(* Logix 5000 project; controller ZaxisVmpEdsSample vendor 1 type 14 code 196 rev 33.11; software revision 33.00 *)

TASK MainTask (continuous, watchdog 500 ms) : MainProgram, Vmp_Interface

MODULES
   Local : vendor 1 type 14 code 196 (5069 0, rev 33.11)
      Inputs : 5069-IB16 (5069 1, rev 2.1, StandardDataDriven RPI 5 ms)
      Outputs : vendor 1 type 7 code 396 (5069 2, rev 2.1, StandardDataDriven RPI 5 ms)
      Vmp_00 : vendor 1449 type 43 code 17 (Ethernet 192.168.2.130, rev 1.4, StandardDataDriven RPI 500 ms)
END_MODULES

TYPE STRING_12 :
STRUCT
   LEN : DINT;
   DATA : SINT[12];
END_STRUCT
END_TYPE

TYPE STRING_16_UDT :
STRUCT
   LEN : DINT;
   DATA : SINT[16];
END_STRUCT
END_TYPE

TYPE STRING_20 :
STRUCT
   LEN : DINT;
   DATA : SINT[20];
END_STRUCT
END_TYPE

TYPE STRING_24 :
STRUCT
   LEN : DINT;
   DATA : SINT[24];
END_STRUCT
END_TYPE

TYPE Vmp_Config :
STRUCT
   CosType : INT;   // Change-of-State Type
   ClassId : INT;   // ClassId
   Instance : INT;   // Instance
   Attribute : INT;   // Attribute
   CfgVersion : INT;   // CfgVersion
   CfgLength : INT;   // CfgLength
   NumberOfHeads : SINT;   // NumberOfHeads
   PumpType : SINT;   // PumpType
   PumpNumber : SINT;   // PumpNumber
   HeadSize : SINT;   // HeadSize
   AdjustStepmode : INT;   // AdjustStepmode
   ZinchRpm : INT;   // ZinchRpm
   Baud : INT;   // Baud
   ExtraSteps : INT;   // ExtraSteps
   SpareInt1 : INT;   // SpareInt1
   SpareInt2 : INT;   // SpareInt2
   ReadyInterlock : BOOL;   // ReadyInterlock
   EthernetRunReady : BOOL;   // EthernetRunReady
   DchpEnabled : BOOL;   // DchpEnabled
   BoreInCm : BOOL;   // BoreInCm
   IoStartFallingEdge : BOOL;   // IoStartFallingEdge
   FullDuplexRs485 : BOOL;   // FullDuplexRs485
   Spare1_6 : BOOL;   // Spare1_6
   IsFinePichAdj : BOOL;   // IsFinePichAdj
   Spare1_8 : BOOL;   // Spare1_8
   Spare1_9 : BOOL;   // Spare1_9
   Spare1_10 : BOOL;   // Spare1_10
   Spare1_11 : BOOL;   // Spare1_11
   Spare1_12 : BOOL;   // Spare1_12
   Spare1_13 : BOOL;   // Spare1_13
   Spare1_14 : BOOL;   // Spare1_14
   Spare1_15 : BOOL;   // Spare1_15
   Spare1_16 : BOOL;   // Spare1_16
   Spare1_17 : BOOL;   // Spare1_17
   Spare1_18 : BOOL;   // Spare1_18
   Spare1_19 : BOOL;   // Spare1_19
   Spare1_20 : BOOL;   // Spare1_20
   Spare1_21 : BOOL;   // Spare1_21
   Spare1_22 : BOOL;   // Spare1_22
   Spare1_23 : BOOL;   // Spare1_23
   IsServo : BOOL;   // IsServo
   OkToResetDevice : BOOL;   // OkToResetDevice
   Spare1_26 : BOOL;   // Spare1_26
   Spare1_27 : BOOL;   // Spare1_27
   Spare1_28 : BOOL;   // Spare1_28
   Spare1_29 : BOOL;   // Spare1_29
   Spare1_30 : BOOL;   // Spare1_30
   Spare1_31 : BOOL;   // Spare1_31
   FirmwareRev : DINT;   // FirmwareRev
   Bore : DINT;   // Bore
   OffsetValue : DINT;   // OffsetValue
   FlashWriteCnt : DINT;   // FlashWriteCnt
   FaultDispenseSensorCnt : DINT;   // FaultDispenseSensorCnt
   FaultDispenseMotorCnt : DINT;   // FaultDispenseMotorCnt
   FaultAdjustSensorCnt : DINT;   // FaultAdjustSensorCnt
   FaultAdjustMotorCnt : DINT;   // FaultAdjustMotorCnt
   SpareDInt1 : DINT;   // SpareDInt1
   SpareDint2 : DINT;   // SpareDint2
   SerialNumber : STRING_16_UDT;   // SerialNumber
   IpAddress : STRING_16_UDT;   // IpAddress
   IpNetmask : STRING_16_UDT;   // IpNetmask
   IpGateway : STRING_16_UDT;   // IpGateway
   MacAddress : STRING_20;   // MacAddress
   ModelNumber : STRING_24;   // ModelNumber
   OptionsAndFittings : STRING_24;   // OptionsAndFittings
   SccsRevDate : STRING_24;   // SccsRevDate
   SccsRev : STRING_12;   // SccsRev
   SccsRevRange : STRING_24;   // SccsRevRange
END_STRUCT
END_TYPE

TYPE VMP_Program :
STRUCT
   CosType : INT;   // CosType
   ClassId : INT;   // ClassId
   Instance : INT;   // Instance
   Attribute : INT;   // Attribute
   CfgVersion : INT;   // CfgVersion
   CfgLength : INT;   // CfgLength
   Direction : BOOL;   // Direction
   ContinuousRun : BOOL;   // ContinuousRun
   Spare1_2 : BOOL;   // Spare1_2
   Spare1_3 : BOOL;   // Spare1_3
   Spare1_4 : BOOL;   // Spare1_4
   Spare1_5 : BOOL;   // Spare1_5
   Spare1_6 : BOOL;   // Spare1_6
   Spare1_7 : BOOL;   // Spare1_7
   Spare1_8 : BOOL;   // Spare1_8
   Spare1_9 : BOOL;   // Spare1_9
   Spare1_10 : BOOL;   // Spare1_10
   Spare1_11 : BOOL;   // Spare1_11
   Spare1_12 : BOOL;   // Spare1_12
   Spare1_13 : BOOL;   // Spare1_13
   Spare1_14 : BOOL;   // Spare1_14
   Spare1_15 : BOOL;   // Spare1_15
   Spare1_16 : BOOL;   // Spare1_16
   Spare1_17 : BOOL;   // Spare1_17
   Spare1_18 : BOOL;   // Spare1_18
   Spare1_19 : BOOL;   // Spare1_19
   Spare1_20 : BOOL;   // Spare1_20
   Spare1_21 : BOOL;   // Spare1_21
   Spare1_22 : BOOL;   // Spare1_22
   Spare1_23 : BOOL;   // Spare1_23
   Spare1_24 : BOOL;   // Spare1_24
   Spare1_25 : BOOL;   // Spare1_25
   Spare1_26 : BOOL;   // Spare1_26
   Spare1_27 : BOOL;   // Spare1_27
   Spare1_28 : BOOL;   // Spare1_28
   Spare1_29 : BOOL;   // Spare1_29
   Spare1_30 : BOOL;   // Spare1_30
   Spare1_31 : BOOL;   // Spare1_31
   ProgramNumber : INT;   // ProgramNumber
   PullBack : INT;   // PullBack
   PullBackRpm : INT;   // PullBackRpm
   PullBackEndCycleRpm : INT;   // PullBackEndCycleRpm
   PullBackEndCycle : INT;   // PullBackEndCycle
   PullBackEndCycleDelay : INT;   // PullBackEndCycleDelay
   InitialRpm : INT;   // InitialRpm
   Rpm : INT;   // Rpm
   FinalRpm : INT;   // FinalRpm
   FineAdjust : INT;   // FineAdjust
   Acceleration : INT;   // Acceleration
   Deceleration : INT;   // Deceleration
   LoopCycles : INT;   // LoopCycles
   LinkedProgram : INT;   // LinkedProgram
   LinkedTimeDelay : INT;   // LinkedTimeDelay
   MotorCurrent : INT;   // MotorCurrent
   Revolutions : INT;   // Revolutions
   PrePumpClamp : INT;   // PrePumpClamp
   PostPumpClamp : INT;   // PostPumpClamp
   AdjInitialRpm : INT;   // AdjInitialRpm
   AdjustRpm : INT;   // AdjustRpm
   AdjustAcceleration : INT;   // AdjustAcceleration
   AdjustDeceleration : INT;   // AdjustDeceleration
   AdjustMotorPwr : INT;   // AdjustMotorPwr
   SpareInt1 : INT;   // SpareInt1
   SpareInt2 : INT;   // SpareInt2
   AdjustMotorSteps : DINT;   // AdjustMotorSteps
   ApproxDispenseTime : DINT;   // ApproxDispenseTime
   Volume : REAL;   // Volume
   SpareDint1 : REAL;   // SpareDint1
   ProgramName : STRING_16_UDT;   // ProgramName
END_STRUCT
END_TYPE

TYPE Vmp_Pump :
STRUCT
   Enabled : BOOL;
   State : INT;   // Current State
   ShotCount : DINT;   // Number of shots
   DisconnectCount : DINT;   // Disconnect Counter
   FaultCount : DINT;   // Fault Counter
   IN : _05A9:VMP_1_4_21408F44:I:0;
   OUT : _05A9:VMP_1_4_0C80E81B:O:0;
   Configuration : Vmp_Config;
   Programs : VMP_Program[50];
   PumpTmr : TIMER;   // Used to time prime and/or zinch mode
END_STRUCT
END_TYPE

TYPE VMP_Setup :
STRUCT
   ReadyInterlock : BOOL;   // RdyInputEnabled
   EthernetRunReady : BOOL;   // EthSendBusy
   HoldOnFault : BOOL;   // HoldOnFault
   Spare1_3 : BOOL;   // Spare Bit
   Spare1_4 : BOOL;   // Spare Bit
   Spare1_5 : BOOL;   // Spare Bit
   Spare1_6 : BOOL;   // Spare Bit
   Spare1_7 : BOOL;   // Spare Bit
   Spare1_8 : BOOL;   // Spare Bit
   Spare1_9 : BOOL;   // Spare Bit
   Spare1_10 : BOOL;   // Spare Bit
   Spare1_11 : BOOL;   // Spare Bit
   Spare1_12 : BOOL;   // Spare Bit
   Spare1_13 : BOOL;   // Spare Bit
   Spare1_14 : BOOL;   // Spare Bit
   Spare1_15 : BOOL;   // Spare Bit
   Spare1_16 : BOOL;   // Spare Bit
   Spare1_17 : BOOL;   // Spare Bit
   Spare1_18 : BOOL;   // Spare Bit
   Spare1_19 : BOOL;   // Spare Bit
   Spare1_20 : BOOL;   // Spare Bit
   Spare1_21 : BOOL;   // Spare Bit
   Spare1_22 : BOOL;   // Spare Bit
   Spare1_23 : BOOL;   // Spare Bit
   Spare1_24 : BOOL;   // Spare Bit
   Spare1_25 : BOOL;   // Spare Bit
   Spare1_26 : BOOL;   // Spare Bit
   Spare1_27 : BOOL;   // Spare Bit
   Spare1_28 : BOOL;   // Spare Bit
   Spare1_29 : BOOL;   // Spare Bit
   Spare1_30 : BOOL;   // Spare Bit
   Spare1_31 : BOOL;   // Spare Bit
   Baud : DINT;   // Baud
   PumpNumber : DINT;   // PumpNumber
   SpareDInt0 : DINT;   // SpareDInt0
   SpareDInt1 : DINT;   // SpareDInt1
   FirmwareRev : REAL;   // FirmRev
   Bore : REAL;   // Bore
   SpareReal0 : REAL;   // SpareReal0
   SpareReal1 : REAL;   // SpareReal1
   SerialNumber : STRING;   // SerialNumber
END_STRUCT
END_TYPE

TYPE VMP_TcpIP_Cfg :
STRUCT
   Status : DINT;   // Status
   Config_Capability : DINT;   // Capability
   Config_Control : DINT;   // IfCtrl
   Path_Size : INT;   // Epath
   Path : SINT[4];   // Padd
   IP_Address : DINT;   // IPAddr
   Network_Address : DINT;   // NetAddr
   Gateway_Address : DINT;   // GateWay
   Name_Server : DINT;   // DNS1
   Name_Server_2 : DINT;   // DNS2
   Domain_Name : STRING;   // Domain
   Host_Name : STRING;   // Host
   Safety_Network_Number : SINT[6];   // Ignore
   TTL : SINT;   // TTL
   Alloc_Control : SINT;   // MultCast
   Reserved : SINT;   // Reserved
   Num_Mcast : INT;   // MultCastAlloc
   Mcast_Start_Addr : DINT;   // MultCastStart
   Selected_Acd : BOOL;   // ACD
   Acd_Activity : SINT;   // ACDState
   Remote_MAC : SINT[6];   // MACRmt
   Arp_Pdu : SINT[28];   // ARP_PDU
   EthernetIP_Quick_Connect : BOOL;   // QuickCon
   Encp_Inactivity_Timeout : INT;   // InactTimeout
END_STRUCT
END_TYPE

ADD_ON_INSTRUCTION Vmp_Run_Pump   (* revision 1.0 *)
VAR_IN_OUT
   Pump : Vmp_Pump; {required}
END_VAR
VAR_INPUT
   State : INT; {required}
   ShotCount : DINT; {required}
   PrimeRevs : DINT; {required}
   ZinchTime : DINT; {required}
END_VAR
VAR
   DirectionONS : BOOL; {access None}
END_VAR

ROUTINE Logic   (* ladder *)
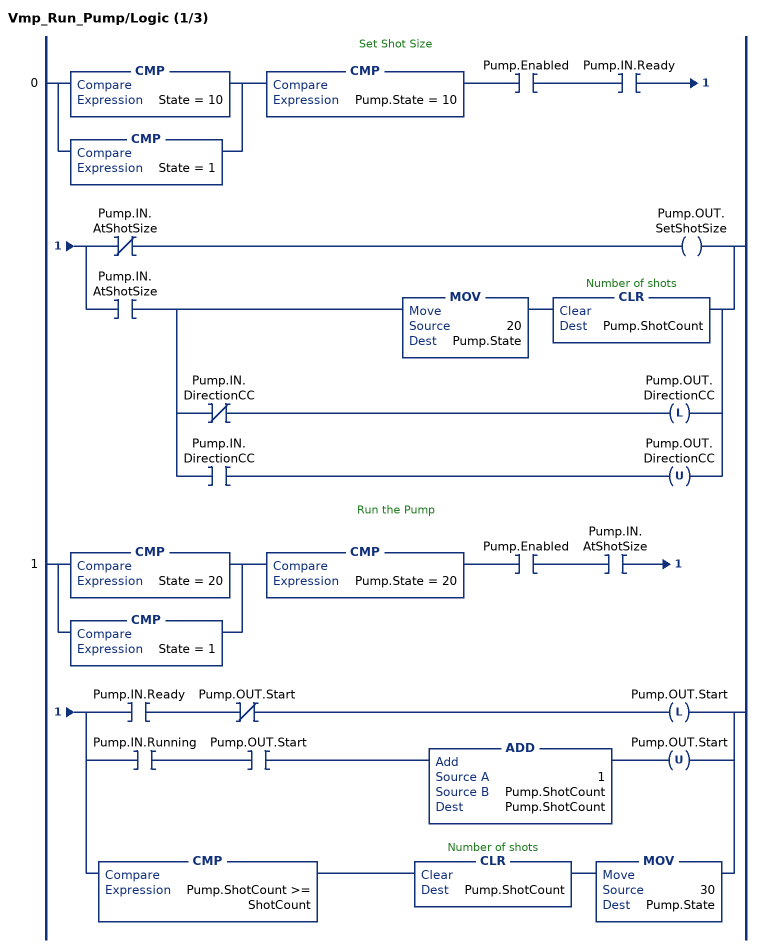
   // Set Shot Size
   0: [CMP(State = 10) ,CMP(State = 1) ]CMP(Pump.State = 10)XIC(Pump.Enabled)XIC(Pump.IN.Ready)[XIO(Pump.IN.AtShotSize) OTE(Pump.OUT.SetShotSize) ,XIC(Pump.IN.AtShotSize) [MOV(20,Pump.State) CLR(Pump.ShotCount) ,XIO(Pump.IN.DirectionCC) OTL(Pump.OUT.DirectionCC) ,XIC(Pump.IN.DirectionCC) OTU(Pump.OUT.DirectionCC) ] ];
   // Run the Pump
   1: [CMP(State = 20) ,CMP(State = 1) ]CMP(Pump.State = 20)XIC(Pump.Enabled)XIC(Pump.IN.AtShotSize)[XIC(Pump.IN.Ready) XIO(Pump.OUT.Start) OTL(Pump.OUT.Start) ,XIC(Pump.IN.Running) XIC(Pump.OUT.Start) ADD(1,Pump.ShotCount,Pump.ShotCount) OTU(Pump.OUT.Start) ,CMP(Pump.ShotCount >= ShotCount) CLR(Pump.ShotCount) MOV(30,Pump.State) ];
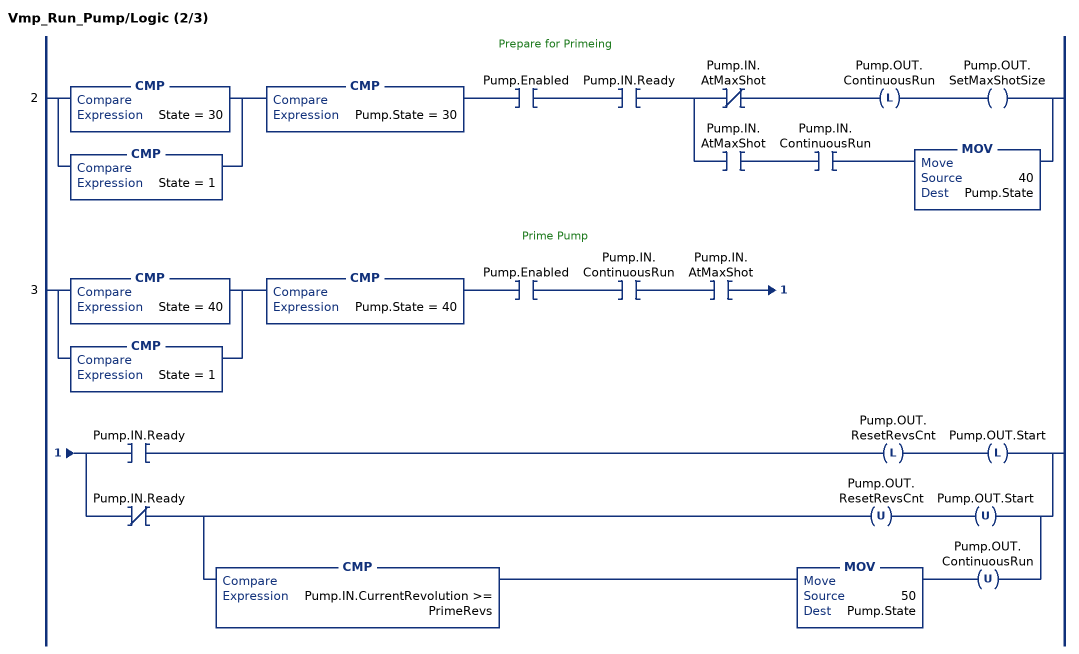
   // Prepare for Primeing
   2: [CMP(State = 30) ,CMP(State = 1) ]CMP(Pump.State = 30)XIC(Pump.Enabled)XIC(Pump.IN.Ready)[XIO(Pump.IN.AtMaxShot) OTL(Pump.OUT.ContinuousRun) OTE(Pump.OUT.SetMaxShotSize) ,XIC(Pump.IN.AtMaxShot) XIC(Pump.IN.ContinuousRun) MOV(40,Pump.State) ];
   // Prime Pump
   3: [CMP(State = 40) ,CMP(State = 1) ]CMP(Pump.State = 40)XIC(Pump.Enabled)XIC(Pump.IN.ContinuousRun)XIC(Pump.IN.AtMaxShot)[XIC(Pump.IN.Ready) OTL(Pump.OUT.ResetRevsCnt) OTL(Pump.OUT.Start) ,XIO(Pump.IN.Ready) [OTU(Pump.OUT.ResetRevsCnt) OTU(Pump.OUT.Start) ,CMP(Pump.IN.CurrentRevolution >= PrimeRevs) MOV(50,Pump.State) OTU(Pump.OUT.ContinuousRun) ] ];
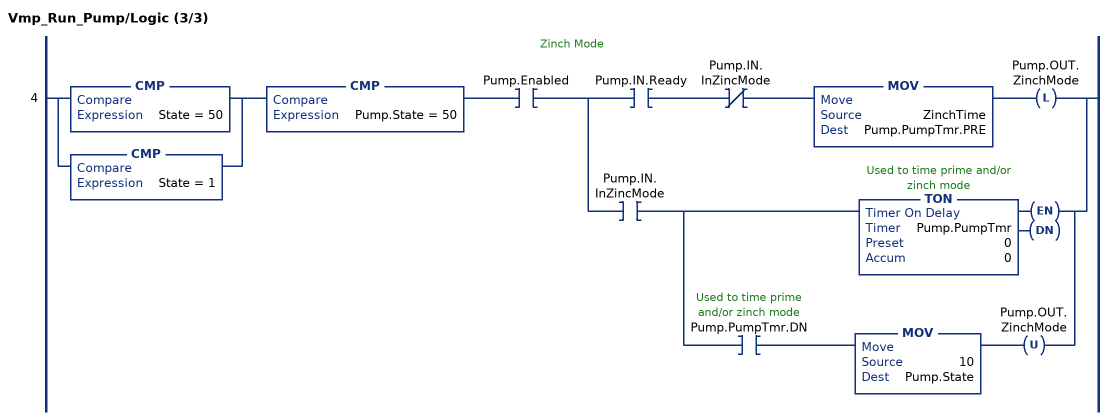
   // Zinch Mode
   4: [CMP(State = 50) ,CMP(State = 1) ]CMP(Pump.State = 50)XIC(Pump.Enabled)[XIC(Pump.IN.Ready) XIO(Pump.IN.InZincMode) MOV(ZinchTime,Pump.PumpTmr.PRE) OTL(Pump.OUT.ZinchMode) ,XIC(Pump.IN.InZincMode) [TON(Pump.PumpTmr,0,0) ,XIC(Pump.PumpTmr.DN) MOV(10,Pump.State) OTU(Pump.OUT.ZinchMode) ] ];
END_ROUTINE
END_ADD_ON_INSTRUCTION

VAR_GLOBAL   (* controller tags *)
   IdleTime : DINT := 3000; {constant}
   PrimeRevs : DINT := 40; {constant}
   ShotCount : DINT := 20; {constant}
   State : INT := 1;
   Vmp_Pumps : Vmp_Pump[1] := ([0].Enabled := 1, [0].State := 10, [0].PumpTmr.PRE := 30000);   // Zaxis Pumps
   VmpConfig_Read : MESSAGE;
        MessageParameters(ServiceCode := 16#0001, DestinationTag := Vmp_Pumps[0].Configuration, ...)
   VmpConfig_Write : MESSAGE;
        MessageParameters(ServiceCode := 16#0002, LocalElement := Vmp_Pumps[0].Configuration, ...)
   VmpProgram_Read : MESSAGE;
        MessageParameters(ServiceCode := 16#0001, DestinationTag := Vmp_Pumps[0].Programs[0], ...)
   VmpProgram_Write : MESSAGE;
        MessageParameters(ServiceCode := 16#0002, LocalElement := Vmp_Pumps[0].Programs[0], ...)
   ZinchTime : DINT := 30000; {constant}
END_VAR

PROGRAM MainProgram   (* main routine MainRoutine *)

ROUTINE MainRoutine   (* ladder *)
END_ROUTINE
END_PROGRAM

PROGRAM Vmp_Interface   (* main routine Vmp_Main *)
VAR
   ChangeBoreSize : BOOL;
   GreenLight : ALIAS FOR Local:2:O.Pt00.Data;
   Init_Button : BOOL;
   Init_ONS : BOOL;
   NumberOfPumps : DINT := 1;
   PumpIdx : DINT;
   Run_EN : BOOL;
   SetBoreSize : BOOL;
   Start_Button : BOOL;
   Stop_Button : BOOL;
   Vmp_Pump_Run : Vmp_Run_Pump := (State := 1, ShotCount := 20, PrimeRevs := 40, ZinchTime := 30000);
   VmpConfig_Read_Do : BOOL;
   VmpConfig_Write_Do : BOOL;
   VmpProgram_Read_Do : BOOL;
   VmpProgram_Write_Do : BOOL;
END_VAR

ROUTINE Vmp_Int   (* ladder *)
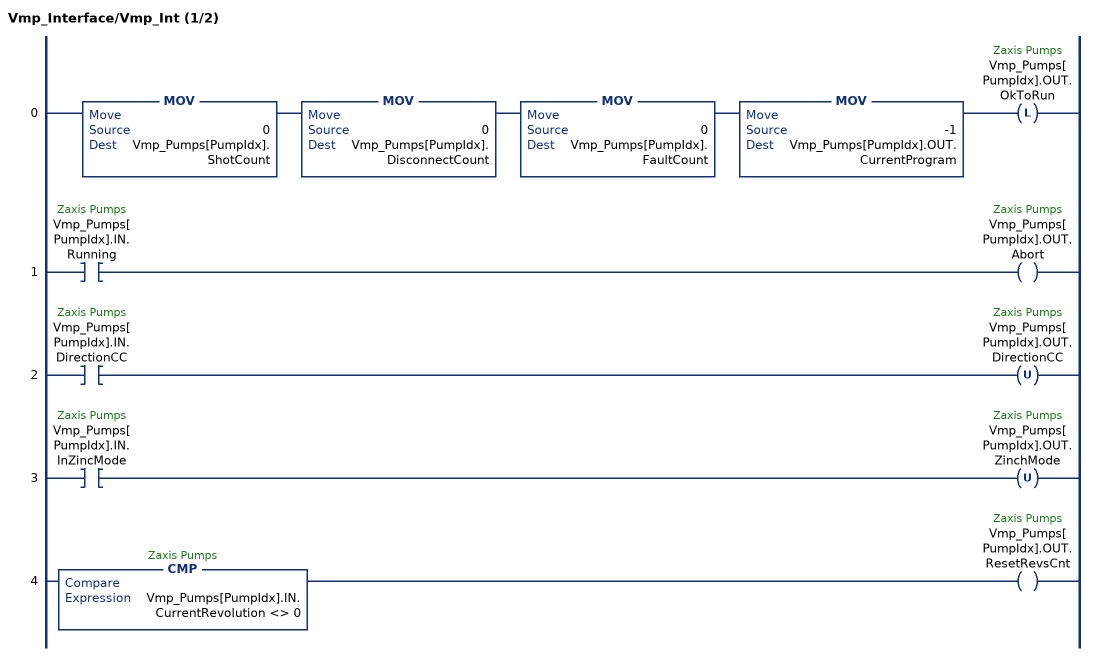
   0: MOV(0,Vmp_Pumps[PumpIdx].ShotCount)MOV(0,Vmp_Pumps[PumpIdx].DisconnectCount)MOV(0,Vmp_Pumps[PumpIdx].FaultCount)MOV(-1,Vmp_Pumps[PumpIdx].OUT.CurrentProgram)OTL(Vmp_Pumps[PumpIdx].OUT.OkToRun);
   1: XIC(Vmp_Pumps[PumpIdx].IN.Running)OTE(Vmp_Pumps[PumpIdx].OUT.Abort);
   2: XIC(Vmp_Pumps[PumpIdx].IN.DirectionCC)OTU(Vmp_Pumps[PumpIdx].OUT.DirectionCC);
   3: XIC(Vmp_Pumps[PumpIdx].IN.InZincMode)OTU(Vmp_Pumps[PumpIdx].OUT.ZinchMode);
   4: CMP(Vmp_Pumps[PumpIdx].IN.CurrentRevolution <> 0)OTE(Vmp_Pumps[PumpIdx].OUT.ResetRevsCnt);
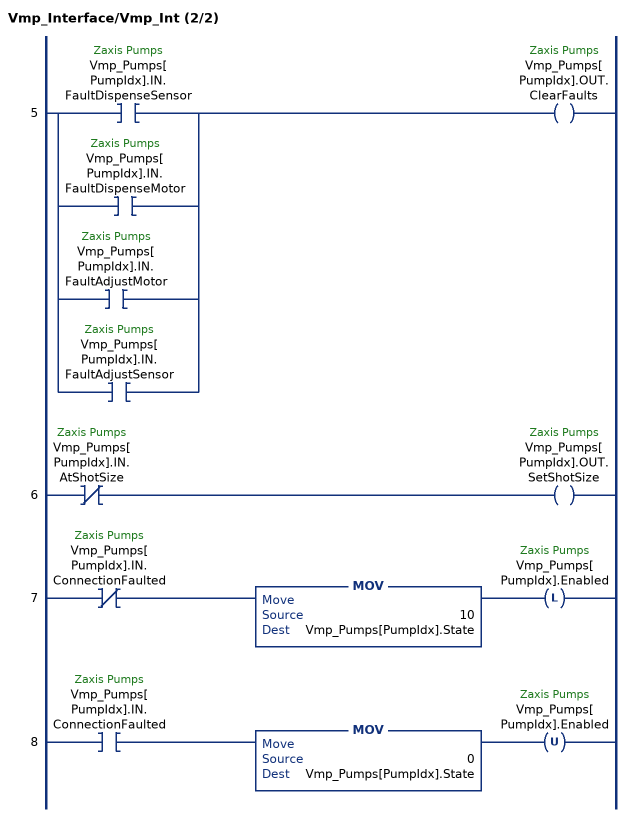
   5: [XIC(Vmp_Pumps[PumpIdx].IN.FaultDispenseSensor) ,XIC(Vmp_Pumps[PumpIdx].IN.FaultDispenseMotor) ,XIC(Vmp_Pumps[PumpIdx].IN.FaultAdjustMotor) ,XIC(Vmp_Pumps[PumpIdx].IN.FaultAdjustSensor) ]OTE(Vmp_Pumps[PumpIdx].OUT.ClearFaults);
   6: XIO(Vmp_Pumps[PumpIdx].IN.AtShotSize)OTE(Vmp_Pumps[PumpIdx].OUT.SetShotSize);
   7: XIO(Vmp_Pumps[PumpIdx].IN.ConnectionFaulted)MOV(10,Vmp_Pumps[PumpIdx].State)OTL(Vmp_Pumps[PumpIdx].Enabled);
   8: XIC(Vmp_Pumps[PumpIdx].IN.ConnectionFaulted)MOV(0,Vmp_Pumps[PumpIdx].State)OTU(Vmp_Pumps[PumpIdx].Enabled);
END_ROUTINE

ROUTINE Vmp_Main   (* ladder *)
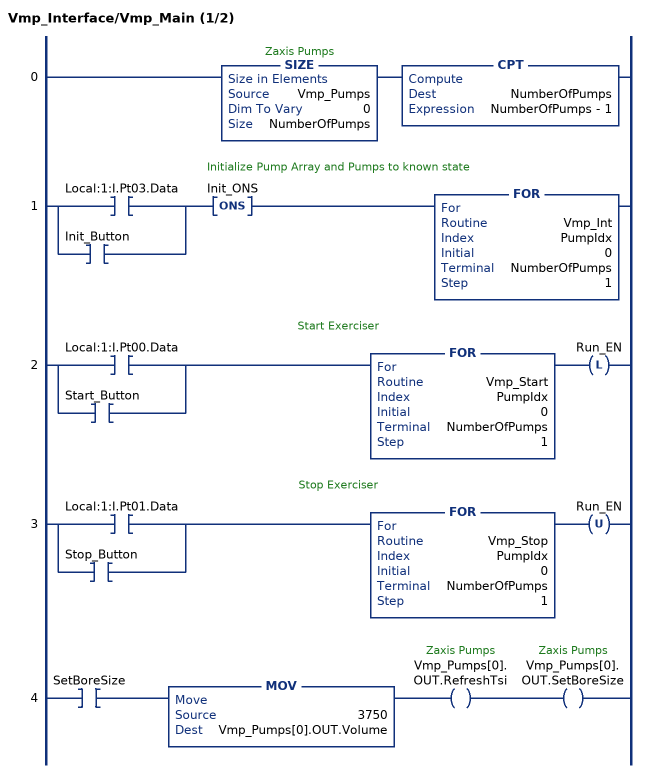
   0: SIZE(Vmp_Pumps,0,NumberOfPumps)CPT(NumberOfPumps,NumberOfPumps - 1);
   // Initialize Pump Array and Pumps to known state
   1: [XIC(Local:1:I.Pt03.Data) ,XIC(Init_Button) ]ONS(Init_ONS)FOR(Vmp_Int,PumpIdx,0,NumberOfPumps,1);
   // Start Exerciser
   2: [XIC(Local:1:I.Pt00.Data) ,XIC(Start_Button) ]FOR(Vmp_Start,PumpIdx,0,NumberOfPumps,1)OTL(Run_EN);
   // Stop Exerciser
   3: [XIC(Local:1:I.Pt01.Data) ,XIC(Stop_Button) ]FOR(Vmp_Stop,PumpIdx,0,NumberOfPumps,1)OTU(Run_EN);
   4: XIC(SetBoreSize)MOV(3750,Vmp_Pumps[0].OUT.Volume)OTE(Vmp_Pumps[0].OUT.RefreshTsi)OTE(Vmp_Pumps[0].OUT.SetBoreSize);
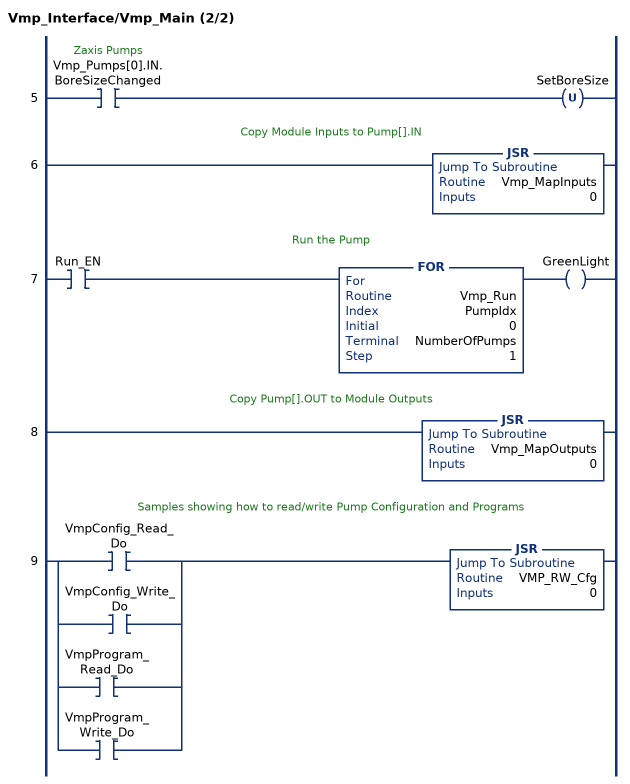
   5: XIC(Vmp_Pumps[0].IN.BoreSizeChanged)OTU(SetBoreSize);
   // Copy Module Inputs to Pump[].IN
   6: JSR(Vmp_MapInputs,0);
   // Run the Pump
   7: XIC(Run_EN)FOR(Vmp_Run,PumpIdx,0,NumberOfPumps,1)OTE(GreenLight);
   // Copy Pump[].OUT to Module Outputs
   8: JSR(Vmp_MapOutputs,0);
   // Samples showing how to read/write Pump Configuration and Programs
   9: [XIC(VmpConfig_Read_Do) ,XIC(VmpConfig_Write_Do) ,XIC(VmpProgram_Read_Do) ,XIC(VmpProgram_Write_Do) ]JSR(VMP_RW_Cfg,0);
END_ROUTINE

ROUTINE Vmp_MapInputs   (* ladder *)
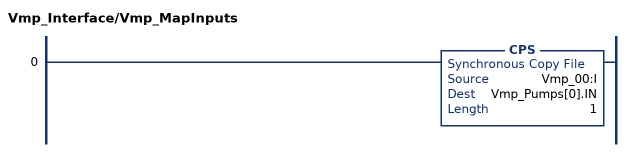
   0: CPS(Vmp_00:I,Vmp_Pumps[0].IN,1);
END_ROUTINE

ROUTINE Vmp_MapOutputs   (* ladder *)
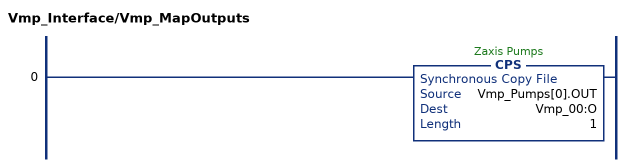
   0: CPS(Vmp_Pumps[0].OUT,Vmp_00:O,1);
END_ROUTINE

ROUTINE Vmp_Run   (* ladder *)
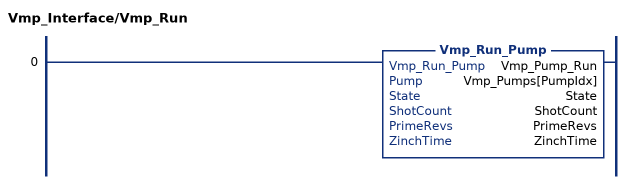
   0: Vmp_Run_Pump(Vmp_Pump_Run,Vmp_Pumps[PumpIdx],State,ShotCount,PrimeRevs,ZinchTime);
END_ROUTINE

ROUTINE VMP_RW_Cfg   (* ladder *)
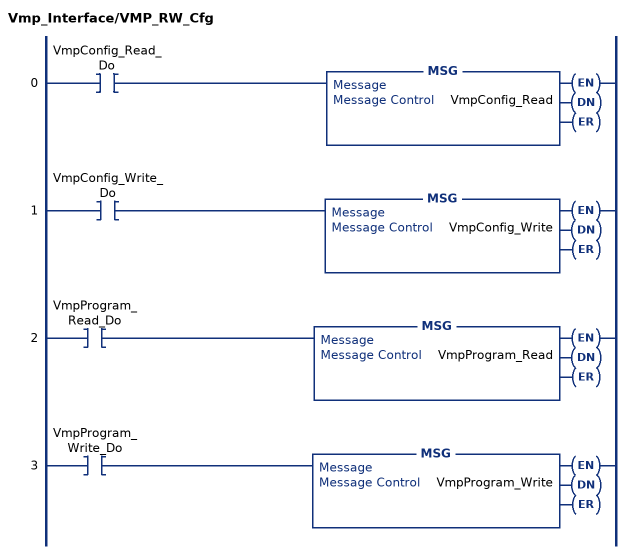
   0: XIC(VmpConfig_Read_Do)MSG(VmpConfig_Read);
   1: XIC(VmpConfig_Write_Do)MSG(VmpConfig_Write);
   2: XIC(VmpProgram_Read_Do)MSG(VmpProgram_Read);
   3: XIC(VmpProgram_Write_Do)MSG(VmpProgram_Write);
END_ROUTINE

ROUTINE Vmp_Start   (* ladder *)
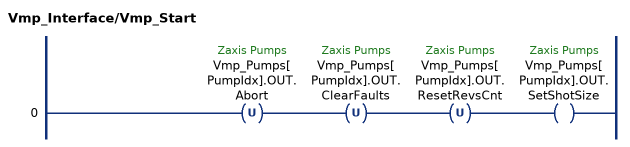
   0: OTU(Vmp_Pumps[PumpIdx].OUT.Abort)OTU(Vmp_Pumps[PumpIdx].OUT.ClearFaults)OTU(Vmp_Pumps[PumpIdx].OUT.ResetRevsCnt)OTE(Vmp_Pumps[PumpIdx].OUT.SetShotSize);
END_ROUTINE

ROUTINE Vmp_Stop   (* ladder *)
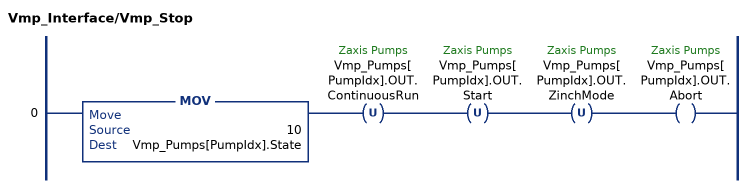
   0: MOV(10,Vmp_Pumps[PumpIdx].State)OTU(Vmp_Pumps[PumpIdx].OUT.ContinuousRun)OTU(Vmp_Pumps[PumpIdx].OUT.Start)OTU(Vmp_Pumps[PumpIdx].OUT.ZinchMode)OTE(Vmp_Pumps[PumpIdx].OUT.Abort);
END_ROUTINE
END_PROGRAM
